// TIA Portal V20 export
TYPE "typeCmControlNodeInterlock"
// stored: Namespace Unit1.Em1
   STRUCT
      unWinder { ExternalWritable := 'False'} : "LER_typeAxisInterlock";
      airShaft { ExternalWritable := 'False'} : "LER_typeTwoWayActuatorInterlock";
      expel { ExternalWritable := 'False'} : "LER_typeTwoWayActuatorInterlock";
   END_STRUCT;
END_TYPE
